Universal Robots PolyScope program: hal.urp

Program hal (installation=default directory=/programs/archive createdIn=5.11.5.1010327 lastSavedIn=5.11.5.1010327 robotSerialNumber=20215500677)
Calibrated DH parameters: a=[0.000204, -0.239222, -0.391845, -0.000001, 0.000022, 0]; d=[0.162722, -355.808559, 353.37206, 2.570385, 0.099741, 0.099629]; alpha=[1.571124, 0.000988, 0.008295, 1.568963, -1.570303, 0]; deltaTheta=[0, -0.973091, 7.204745, 0.05153, 0, 0]
Robot Program (runOnlyOnce=true)
  Script file /programs/usbdisk_0/Move.script
    | def Move() :
    | set_target_payload(1.290000, [0.000000, -0.007000, 0.042000], [0.002353, 0.002353, 0.002353, 0.000000, 0.000000, 0.000000])
    | set_tcp(p[0,0,0,0,0,0])
    | movej([1.936402,-1.198617,-1.58622,-1.927552,1.570796,3.507198], a=1, v=1)
    | movej([0.417377,-2.271868,-0.828392,-1.612128,1.570796,1.988173], a=1, v=1)
    | movej([0.738069,-1.436084,-1.911521,-1.364784,1.570796,2.308865], a=1, v=1)
    | 
    | end
    | 
    | 
    | Move()
